// SIMATIC S7-200 project (STEP 7-Micro/WIN), CPU 224 REL 01.11

SYMBOL_TABLE USER1
A1               Q0.0
A2               Q0.2
B1               Q0.1
B2               Q0.3
ONN              I0.0
OFF              I0.1
END_SYMBOL_TABLE

ORGANIZATION_BLOCK MAIN:OB1
TITLE=PROGRAM COMMENTS
BEGIN
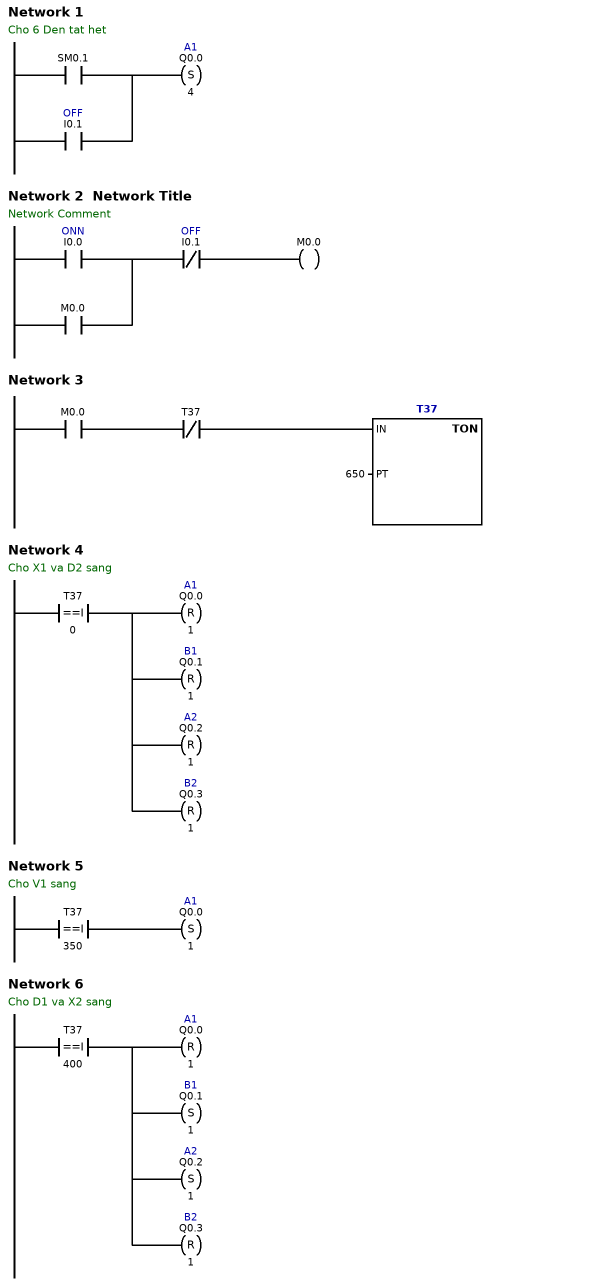
Network 1
// Cho 6 Den tat het
// (network saved uncompiled; LAD cells follow)
// row 0: c0 -| |- SM0.1 v  c1 -(S) A1:Q0.0, 4
// row 1: c0 -| |- OFF:I0.1 ^
Network 2 // Network Title
// Network Comment
LD     ONN:I0.0
O      M0.0
AN     OFF:I0.1
=      M0.0
Network 3
// (network saved uncompiled; LAD cells follow)
// row 0: c0 -| |- M0.0  c1 -|/|- T37  c2 --  c3 [TON T37 IN:=power@row0, PT:=650]
// row 1: c3 [box]
Network 4
// Cho X1 va D2 sang
// (network saved uncompiled; LAD cells follow)
// row 0: c0 -|==I|- T37, 0 v  c1 -(R) A1:Q0.0, 1
// row 1: c0 ^v  c1 -(R) B1:Q0.1, 1
// row 2: c0 ^v  c1 -(R) A2:Q0.2, 1
// row 3: c0 ^  c1 -(R) B2:Q0.3, 1
Network 5
// Cho V1 sang
LDW=   T37, 350
S      A1:Q0.0, 1
Network 6
// Cho D1 va X2 sang
// (network saved uncompiled; LAD cells follow)
// row 0: c0 -|==I|- T37, 400 v  c1 -(R) A1:Q0.0, 1
// row 1: c0 ^v  c1 -(S) B1:Q0.1, 1
// row 2: c0 ^v  c1 -(S) A2:Q0.2, 1
// row 3: c0 ^  c1 -(R) B2:Q0.3, 1
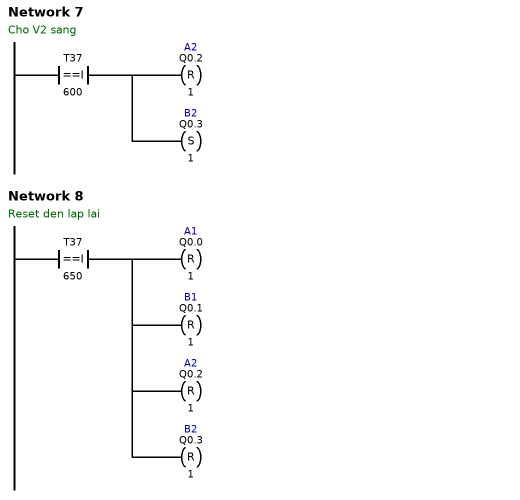
Network 7
// Cho V2 sang
// (network saved uncompiled; LAD cells follow)
// row 0: c0 -|==I|- T37, 600 v  c1 -(R) A2:Q0.2, 1
// row 1: c0 ^  c1 -(S) B2:Q0.3, 1
Network 8
// Reset den lap lai 
// (network saved uncompiled; LAD cells follow)
// row 0: c0 -|==I|- T37, 650 v  c1 -(R) A1:Q0.0, 1
// row 1: c0 ^v  c1 -(R) B1:Q0.1, 1
// row 2: c0 ^v  c1 -(R) A2:Q0.2, 1
// row 3: c0 ^  c1 -(R) B2:Q0.3, 1
END_ORGANIZATION_BLOCK
